{attribute 'linkalways'} 
{attribute 'no_explicit_call' := 'This FB is a CLASS and must be accessed using methods or properties'}
{attribute 'enable_dynamic_creation'}
FUNCTION_BLOCK Node_ContainerType_Vector_Vector_LREAL EXTENDS Node
VAR
    out : _GUID;
END_VAR

METHOD PUBLIC  Clone : I_Node
VAR
	pNode : POINTER TO Node_ContainerType_Vector_Vector_LREAL;
END_VAR
pNode := __NEW(Node_ContainerType_Vector_Vector_LREAL);
Clone := pNode^;
END_METHOD

METHOD FB_init : BOOL
VAR_INPUT
	bInitRetains : BOOL; // if TRUE, the retain variables are initialized (warm start / cold start)
	bInCopyCode : BOOL;  // if TRUE, the instance afterwards gets moved into the copy code (online change)
END_VAR
AddOutput('out', out);
END_METHOD

METHOD PROTECTED OnExecute
out.Value := ContainerType_Vector_Vector_LREAL;
END_METHOD

END_FUNCTION_BLOCK

(* stored: Version 1.1.0.1, ProductVersion 3.1.4026.17
   POU Node_ContainerType_Vector_Vector_LREAL: Id {8e741521-437e-0d82-1c43-8ed13fff3d2b}, SpecialFunc None
   Folder Constructor: Id {1e0ca8f9-4947-0ffb-13ec-8b2f1671f5bb}
   Method Clone: Id {21791ec8-fac0-0ce8-0a72-7ed3635097d7}
   Method FB_init: Id {f8c41e98-af22-0da0-3e29-13dc656ed9a4}
   Method OnExecute: Id {aa233b11-b31e-0681-03c5-58fbba826a62} *)
